{attribute 'Tc2GvlVarNames'}
VAR_GLOBAL RETAIN

END_VAR

(* stored: Version 1.1.0.1, ProductVersion 3.1.4022.7
   GVL Setup_Data_1: Id {8ae1fcbf-0109-4bfc-9a34-37364020ba6a} *)
